(* CODESYS project ProximitySensor.xml

Project tree, tasks and I/O mapping:
  function block ProximitySensor [LD]
*)

// ProximitySensor
FUNCTION_BLOCK ProximitySensor
// The proximity sensor function block represents proximity sensor functionality. 
// When the sensor sees its target this function block will output to Q after the OnDelay time has passed,
// and will continue to output until the sensor no longer sees its target, AND the OffDelay time has passed.
VAR_INPUT
	IN: 				BOOL;				//
	OnDelay: 			TIME;				//
	OffDelay: 			TIME;				//
END_VAR
VAR_OUTPUT
	Q: 					BOOL;				//
END_VAR
VAR
	_OnDelayTimer: 		TON;				//
	_OffDelayTimer: 	TON;				//
END_VAR

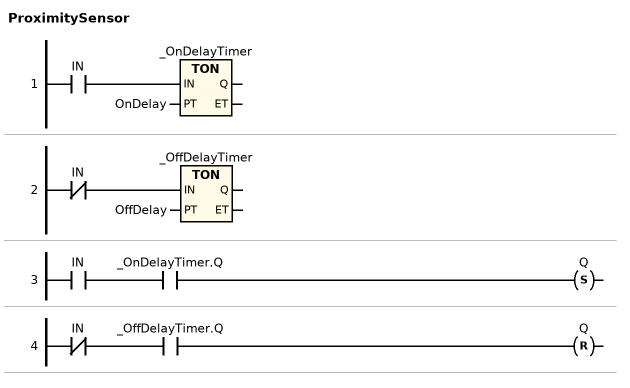
// NETWORK 1
_OnDelayTimer(IN := IN, PT := OnDelay); // TON

// NETWORK 2
_OffDelayTimer(IN := NOT IN, PT := OffDelay); // TON

// NETWORK 3
Q S= IN AND _OnDelayTimer.Q;

// NETWORK 4
Q R= NOT IN AND _OffDelayTimer.Q;

END_FUNCTION_BLOCK
